Staubli VAL3: buildList.pgx

program buildList()
  local num l_nSize
  local string l_sEvent
  local num i
  local string l_sProg
  local num l_nDone
  local num l_nTotal
  local num l_nType
  local string l_sItem
begin
  // INIT the list
  l_sItem=""
  call use:stringCopy(l_sItem,sList)
  // Build the list
  call processList:getDefaultType(l_nType)
  call processList:getSize(l_nSize,l_nType)
  if l_nSize>0
    for i=0 to (l_nSize-1)
      call processList:getCycle(l_sProg,l_nTotal,l_nDone,i,l_nType)
      if l_sProg!=""
        l_sEvent=(" ["+toString("1",l_nDone)+"/"+toString("1",l_nTotal)+"]")
        call listAdd(toString("2",i+1)+" "+l_sProg+l_sEvent)
      endIf
    endFor
  endIf
end
